// TIA Portal V20 export
DATA_BLOCK "LBP_ParamAlarmMsgs"   // DB5
TITLE = PLC-Error / Messages / Erreur AP / messages
{ S7_Optimized_Access := 'FALSE' }
AUTHOR : SINUMERIK
FAMILY : SINUMERIK_ONE
VERSION : 6.24
// Interface between user program and LBP_GenAlarmMsgs [FC10], contains the parameter assignment of the alarms for the bit arrays in the LBP_AlarmMsgs [DB2] as fault or status message. / Interface entre programme utilisateur et LBP_GenAlarmMsgs [FC10] contient l'affectation de paramètres des alarmes pour les tableaux de bits dans LBP_AlarmMsgs [DB2]  en tant que signalisations de défaut et d'état.
// stored: AutoNumber false
   VAR RETAIN
      Ch1_DB2_310 : Bool := TRUE;   // (Channels 1-10, 18 bits each): DB2.DBB310; error messages / (Canaux 1-10, 18 bits chacun) : DB2.DBB310 ; signalisations de défaut
      Ch1_DB2_311 : Bool := FALSE;   // Channel 1, DB2.DBB311; operating messages / Canal 1, DB2.DBB311 ; signalisations d'état
      Ch1_DB2_312 : Bool := TRUE;   // Channel 1, DB2.DBB312; error messages / Canal 1, DB2.DBB312 ; signalisations de défaut
      Ch1_DB2_313 : Bool := TRUE;   // Error messages / Signalisations de défaut
      Ch1_DB2_314 : Bool := FALSE;   // Operating messages / Signalisations d'état
      Ch1_DB2_315 : Bool := FALSE;   // Operating messages / Signalisations d'état
      Ch1_DB2_316 : Bool := TRUE;   // Error messages / Signalisations de défaut
      Ch1_DB2_317 : Bool := TRUE;   // Error messages / Signalisations de défaut
      Ch1_DB2_318 : Bool := FALSE;   // Operating messages / Signalisations d'état
      Ch1_DB2_319 : Bool := FALSE;   // Operating messages / Signalisations d'état
      Ch1_DB2_320 : Bool := TRUE;   // Error messages / Signalisations de défaut
      Ch1_DB2_321 : Bool := FALSE;   // Operating messages / Signalisations d'état
      Ch1_DB2_322 : Bool := TRUE;   // Error messages / Signalisations de défaut
      Ch1_DB2_323 : Bool := FALSE;   // Operating messages / Signalisations d'état
      Ch1_DB2_324 : Bool := TRUE;   // Error messages / Signalisations de défaut
      Ch1_DB2_325 : Bool := FALSE;   // Operating messages / Signalisations d'état
      Ch1_DB2_326 : Bool := TRUE;   // Error messages / Signalisations de défaut
      Ch1_DB2_327 : Bool := FALSE;   // Operating messages / Signalisations d'état
      Ch2_DB2_328 : Bool := TRUE;   // Channel 2, DB2.DBB328; error messages / Canal 2, DB2.DBB328 ; signalisations de défaut
      Ch2_DB2_329 : Bool := FALSE;   // Channel 2, DB2.DBB329; operating messages / Canal 2, DB2.DBB329 ; signalisations d'état
      Ch2_DB2_330 : Bool := TRUE;   // Error messages / Signalisations de défaut
      Ch2_DB2_331 : Bool := TRUE;   // Error messages / Signalisations de défaut
      Ch2_DB2_332 : Bool := FALSE;   // Operating messages / Signalisations d'état
      Ch2_DB2_333 : Bool := FALSE;   // Operating messages / Signalisations d'état
      Ch2_DB2_334 : Bool := TRUE;   // Error messages / Signalisations de défaut
      Ch2_DB2_335 : Bool := TRUE;   // Error messages / Signalisations de défaut
      Ch2_DB2_336 : Bool := FALSE;   // Operating messages / Signalisations d'état
      Ch2_DB2_337 : Bool := FALSE;   // Operating messages / Signalisations d'état
      Ch2_DB2_338 : Bool := TRUE;   // Error messages / Signalisations de défaut
      Ch2_DB2_339 : Bool := FALSE;   // Operating messages / Signalisations d'état
      Ch2_DB2_340 : Bool := TRUE;   // Error messages / Signalisations de défaut
      Ch2_DB2_341 : Bool := FALSE;   // Operating messages / Signalisations d'état
      Ch2_DB2_342 : Bool := TRUE;   // Error messages / Signalisations de défaut
      Ch2_DB2_343 : Bool := FALSE;   // Operating messages / Signalisations d'état
      Ch2_DB2_344 : Bool := TRUE;   // Error messages / Signalisations de défaut
      Ch2_DB2_345 : Bool := FALSE;   // Operating messages / Signalisations d'état
      Ch3_DB2_346 : Bool := TRUE;   // Channel 3, DB2.DBB346; error messages / Canal 3, DB2.DBB346 ; signalisations de défaut
      Ch3_DB2_347 : Bool := FALSE;   // Channel 3, DB2.DBB347; operating messages / Canal 3, DB2.DBB347 ; signalisations d'état
      Ch3_DB2_348 : Bool := TRUE;   // Error messages / Signalisations de défaut
      Ch3_DB2_349 : Bool := TRUE;   // Error messages / Signalisations de défaut
      Ch3_DB2_350 : Bool := FALSE;   // Operating messages / Signalisations d'état
      Ch3_DB2_351 : Bool := FALSE;   // Operating messages / Signalisations d'état
      Ch3_DB2_352 : Bool := TRUE;   // Error messages / Signalisations de défaut
      Ch3_DB2_353 : Bool := TRUE;   // Error messages / Signalisations de défaut
      Ch3_DB2_354 : Bool := FALSE;   // Operating messages / Signalisations d'état
      Ch3_DB2_355 : Bool := FALSE;   // Operating messages / Signalisations d'état
      Ch3_DB2_356 : Bool := TRUE;   // Error messages / Signalisations de défaut
      Ch3_DB2_357 : Bool := FALSE;   // Operating messages / Signalisations d'état
      Ch3_DB2_358 : Bool := TRUE;   // Error messages / Signalisations de défaut
      Ch3_DB2_359 : Bool := FALSE;   // Operating messages / Signalisations d'état
      Ch3_DB2_360 : Bool := TRUE;   // Error messages / Signalisations de défaut
      Ch3_DB2_361 : Bool := FALSE;   // Operating messages / Signalisations d'état
      Ch3_DB2_362 : Bool := TRUE;   // Error messages / Signalisations de défaut
      Ch3_DB2_363 : Bool := FALSE;   // Operating messages / Signalisations d'état
      Ch4_DB2_364 : Bool := TRUE;   // Channel 4, DB2.DBB364; error messages / Canal 4, DB2.DBB364 ; signalisations de défaut
      Ch4_DB2_365 : Bool := FALSE;   // Channel 4, DB2.DBB365; operating messages / Canal 4, DB2.DBB365 ; signalisations d'état
      Ch4_DB2_366 : Bool := TRUE;   // Error messages / Signalisations de défaut
      Ch4_DB2_367 : Bool := TRUE;   // Error messages / Signalisations de défaut
      Ch4_DB2_368 : Bool := FALSE;   // Operating messages / Signalisations d'état
      Ch4_DB2_369 : Bool := FALSE;   // Operating messages / Signalisations d'état
      Ch4_DB2_370 : Bool := TRUE;   // Error messages / Signalisations de défaut
      Ch4_DB2_371 : Bool := TRUE;   // Error messages / Signalisations de défaut
      Ch4_DB2_372 : Bool := FALSE;   // Operating messages / Signalisations d'état
      Ch4_DB2_373 : Bool := FALSE;   // Operating messages / Signalisations d'état
      Ch4_DB2_374 : Bool := TRUE;   // Error messages / Signalisations de défaut
      Ch4_DB2_375 : Bool := FALSE;   // Operating messages / Signalisations d'état
      Ch4_DB2_376 : Bool := TRUE;   // Error messages / Signalisations de défaut
      Ch4_DB2_377 : Bool := FALSE;   // Operating messages / Signalisations d'état
      Ch4_DB2_378 : Bool := TRUE;   // Error messages / Signalisations de défaut
      Ch4_DB2_379 : Bool := FALSE;   // Operating messages / Signalisations d'état
      Ch4_DB2_380 : Bool := TRUE;   // Error messages / Signalisations de défaut
      Ch4_DB2_381 : Bool := FALSE;   // Operating messages / Signalisations d'état
      Ch5_DB2_382 : Bool := TRUE;   // Channel 5, DB2.DBB382; error messages / Canal 5, DB2.DBB382 ; signalisations de défaut
      Ch5_DB2_383 : Bool := FALSE;   // Channel 5, DB2.DBB383; operating messages / Canal 5, DB2.DBB383 ; signalisations d'état
      Ch5_DB2_384 : Bool := TRUE;   // Error messages / Signalisations de défaut
      Ch5_DB2_385 : Bool := TRUE;   // Error messages / Signalisations de défaut
      Ch5_DB2_386 : Bool := FALSE;   // Operating messages / Signalisations d'état
      Ch5_DB2_387 : Bool := FALSE;   // Operating messages / Signalisations d'état
      Ch5_DB2_388 : Bool := TRUE;   // Error messages / Signalisations de défaut
      Ch5_DB2_389 : Bool := TRUE;   // Error messages / Signalisations de défaut
      Ch5_DB2_390 : Bool := FALSE;   // Operating messages / Signalisations d'état
      Ch5_DB2_391 : Bool := FALSE;   // Operating messages / Signalisations d'état
      Ch5_DB2_392 : Bool := TRUE;   // Error messages / Signalisations de défaut
      Ch5_DB2_393 : Bool := FALSE;   // Operating messages / Signalisations d'état
      Ch5_DB2_394 : Bool := TRUE;   // Error messages / Signalisations de défaut
      Ch5_DB2_395 : Bool := FALSE;   // Operating messages / Signalisations d'état
      Ch5_DB2_396 : Bool := TRUE;   // Error messages / Signalisations de défaut
      Ch5_DB2_397 : Bool := FALSE;   // Operating messages / Signalisations d'état
      Ch5_DB2_398 : Bool := TRUE;   // Error messages / Signalisations de défaut
      Ch5_DB2_399 : Bool := FALSE;   // Operating messages / Signalisations d'état
      Ch6_DB2_400 : Bool := TRUE;   // Channel 6, DB2.DBB400; error messages / Canal 6, DB2.DBB400 ; signalisations de défaut
      Ch6_DB2_401 : Bool := FALSE;   // Channel 6, DB2.DBB401; operating messages / Canal 6, DB2.DBB401 ; signalisations d'état
      Ch6_DB2_402 : Bool := TRUE;   // Error messages / Signalisations de défaut
      Ch6_DB2_403 : Bool := TRUE;   // Error messages / Signalisations de défaut
      Ch6_DB2_404 : Bool := FALSE;   // Operating messages / Signalisations d'état
      Ch6_DB2_405 : Bool := FALSE;   // Operating messages / Signalisations d'état
      Ch6_DB2_406 : Bool := TRUE;   // Error messages / Signalisations de défaut
      Ch6_DB2_407 : Bool := TRUE;   // Error messages / Signalisations de défaut
      Ch6_DB2_408 : Bool := FALSE;   // Operating messages / Signalisations d'état
      Ch6_DB2_409 : Bool := FALSE;   // Operating messages / Signalisations d'état
      Ch6_DB2_410 : Bool := TRUE;   // Error messages / Signalisations de défaut
      Ch6_DB2_411 : Bool := FALSE;   // Operating messages / Signalisations d'état
      Ch6_DB2_412 : Bool := TRUE;   // Error messages / Signalisations de défaut
      Ch6_DB2_413 : Bool := FALSE;   // Operating messages / Signalisations d'état
      Ch6_DB2_414 : Bool := TRUE;   // Error messages / Signalisations de défaut
      Ch6_DB2_415 : Bool := FALSE;   // Operating messages / Signalisations d'état
      Ch6_DB2_416 : Bool := TRUE;   // Error messages / Signalisations de défaut
      Ch6_DB2_417 : Bool := FALSE;   // Operating messages / Signalisations d'état
      Ch7_DB2_418 : Bool := TRUE;   // Channel 7, DB2.DBB418; error messages / Canal 7, DB2.DBB418 ; signalisations de défaut
      Ch7_DB2_419 : Bool := FALSE;   // Channel 7, DB2.DBB419; operating messages / Canal 7, DB2.DBB419 ; signalisations d'état
      Ch7_DB2_420 : Bool := TRUE;   // Error messages / Signalisations de défaut
      Ch7_DB2_421 : Bool := TRUE;   // Error messages / Signalisations de défaut
      Ch7_DB2_422 : Bool := FALSE;   // Operating messages / Signalisations d'état
      Ch7_DB2_423 : Bool := FALSE;   // Operating messages / Signalisations d'état
      Ch7_DB2_424 : Bool := TRUE;   // Error messages / Signalisations de défaut
      Ch7_DB2_425 : Bool := TRUE;   // Error messages / Signalisations de défaut
      Ch7_DB2_426 : Bool := FALSE;   // Operating messages / Signalisations d'état
      Ch7_DB2_427 : Bool := FALSE;   // Operating messages / Signalisations d'état
      Ch7_DB2_428 : Bool := TRUE;   // Error messages / Signalisations de défaut
      Ch7_DB2_429 : Bool := FALSE;   // Operating messages / Signalisations d'état
      Ch7_DB2_430 : Bool := TRUE;   // Error messages / Signalisations de défaut
      Ch7_DB2_431 : Bool := FALSE;   // Operating messages / Signalisations d'état
      Ch7_DB2_432 : Bool := TRUE;   // Error messages / Signalisations de défaut
      Ch7_DB2_433 : Bool := FALSE;   // Operating messages / Signalisations d'état
      Ch7_DB2_434 : Bool := TRUE;   // Error messages / Signalisations de défaut
      Ch7_DB2_435 : Bool := FALSE;   // Operating messages / Signalisations d'état
      Ch8_DB2_436 : Bool := TRUE;   // Channel 8, DB2.DBB436; error messages / Canal 8, DB2.DBB436 ; signalisations de défaut
      Ch8_DB2_437 : Bool := FALSE;   // Channel 8, DB2.DBB437; operating messages / Canal 8, DB2.DBB437 ; signalisations d'état
      Ch8_DB2_438 : Bool := TRUE;   // Error messages / Signalisations de défaut
      Ch8_DB2_439 : Bool := TRUE;   // Error messages / Signalisations de défaut
      Ch8_DB2_440 : Bool := FALSE;   // Operating messages / Signalisations d'état
      Ch8_DB2_441 : Bool := FALSE;   // Operating messages / Signalisations d'état
      Ch8_DB2_442 : Bool := TRUE;   // Error messages / Signalisations de défaut
      Ch8_DB2_443 : Bool := TRUE;   // Error messages / Signalisations de défaut
      Ch8_DB2_444 : Bool := FALSE;   // Operating messages / Signalisations d'état
      Ch8_DB2_445 : Bool := FALSE;   // Operating messages / Signalisations d'état
      Ch8_DB2_446 : Bool := TRUE;   // Error messages / Signalisations de défaut
      Ch8_DB2_447 : Bool := FALSE;   // Operating messages / Signalisations d'état
      Ch8_DB2_448 : Bool := TRUE;   // Error messages / Signalisations de défaut
      Ch8_DB2_449 : Bool := FALSE;   // Operating messages / Signalisations d'état
      Ch8_DB2_450 : Bool := TRUE;   // Error messages / Signalisations de défaut
      Ch8_DB2_451 : Bool := FALSE;   // Operating messages / Signalisations d'état
      Ch8_DB2_452 : Bool := TRUE;   // Error messages / Signalisations de défaut
      Ch8_DB2_453 : Bool := FALSE;   // Operating messages / Signalisations d'état
      Ch9_DB2_454 : Bool := TRUE;   // Channel 9, DB2.DBB454; error messages / Canal 9, DB2.DBB454 ; signalisations de défaut
      Ch9_DB2_455 : Bool := FALSE;   // Channel 9, DB2.DBB455; operating messages / Canal 9, DB2.DBB455 ; signalisations d'état
      Ch9_DB2_456 : Bool := TRUE;   // Error messages / Signalisations de défaut
      Ch9_DB2_457 : Bool := TRUE;   // Error messages / Signalisations de défaut
      Ch9_DB2_458 : Bool := FALSE;   // Operating messages / Signalisations d'état
      Ch9_DB2_459 : Bool := FALSE;   // Operating messages / Signalisations d'état
      Ch9_DB2_460 : Bool := TRUE;   // Error messages / Signalisations de défaut
      Ch9_DB2_461 : Bool := TRUE;   // Error messages / Signalisations de défaut
      Ch9_DB2_462 : Bool := FALSE;   // Operating messages / Signalisations d'état
      Ch9_DB2_463 : Bool := FALSE;   // Operating messages / Signalisations d'état
      Ch9_DB2_464 : Bool := TRUE;   // Error messages / Signalisations de défaut
      Ch9_DB2_465 : Bool := FALSE;   // Operating messages / Signalisations d'état
      Ch9_DB2_466 : Bool := TRUE;   // Error messages / Signalisations de défaut
      Ch9_DB2_467 : Bool := FALSE;   // Operating messages / Signalisations d'état
      Ch9_DB2_468 : Bool := TRUE;   // Error messages / Signalisations de défaut
      Ch9_DB2_469 : Bool := FALSE;   // Operating messages / Signalisations d'état
      Ch9_DB2_470 : Bool := TRUE;   // Error messages / Signalisations de défaut
      Ch9_DB2_471 : Bool := FALSE;   // Operating messages / Signalisations d'état
      Ch10_DB2_472 : Bool := TRUE;   // Channel 10, DB2.DBB472; error messages / Canal 10, DB2.DBB472 ; signalisations de défaut
      Ch10_DB2_473 : Bool := FALSE;   // Channel 10, DB2.DBB473; operating messages / Canal 10, DB2.DBB473 ; signalisations d'état
      Ch10_DB2_474 : Bool := TRUE;   // Error messages / Signalisations de défaut
      Ch10_DB2_475 : Bool := TRUE;   // Error messages / Signalisations de défaut
      Ch10_DB2_476 : Bool := FALSE;   // Operating messages / Signalisations d'état
      Ch10_DB2_477 : Bool := FALSE;   // Operating messages / Signalisations d'état
      Ch10_DB2_478 : Bool := TRUE;   // Error messages / Signalisations de défaut
      Ch10_DB2_479 : Bool := TRUE;   // Error messages / Signalisations de défaut
      Ch10_DB2_480 : Bool := FALSE;   // Operating messages / Signalisations d'état
      Ch10_DB2_481 : Bool := FALSE;   // Operating messages / Signalisations d'état
      Ch10_DB2_482 : Bool := TRUE;   // Error messages / Signalisations de défaut
      Ch10_DB2_483 : Bool := FALSE;   // Operating messages / Signalisations d'état
      Ch10_DB2_484 : Bool := TRUE;   // Error messages / Signalisations de défaut
      Ch10_DB2_485 : Bool := FALSE;   // Operating messages / Signalisations d'état
      Ch10_DB2_486 : Bool := TRUE;   // Error messages / Signalisations de défaut
      Ch10_DB2_487 : Bool := FALSE;   // Operating messages / Signalisations d'état
      Ch10_DB2_488 : Bool := TRUE;   // Error messages / Signalisations de défaut
      Ch10_DB2_489 : Bool := FALSE;   // Operating messages / Signalisations d'état
      Ax1_DB2_490 : Bool := TRUE;   // (Axes/Spindles 1-31, 2 bits each): DB2.DBB490; error messages / (Axes/broches 1-31, 2 bits chacun) : DB2.DBB490 ; signalisations de défaut
      Ax1_DB2_491 : Bool := FALSE;   // Axis/Spindle 1, DB2.DBB491; operating messages / Axe/broche 1, DB2.DBB491 ; signalisations d'état
      Ax2_DB2_492 : Bool := TRUE;   // Axis/Spindle 2, DB2.DBB492; error messages / Axe/broche 2, DB2.DBB492 ; signalisations de défaut
      Ax2_DB2_493 : Bool := FALSE;   // Axis/Spindle 2, DB2.DBB493; operating messages / Axe/broche 2, DB2.DBB493 ; signalisations d'état
      Ax3_DB2_494 : Bool := TRUE;   // Error messages / Signalisations de défaut
      Ax3_DB2_495 : Bool := FALSE;   // Operating messages / Signalisations d'état
      Ax4_DB2_496 : Bool := TRUE;   // Error messages / Signalisations de défaut
      Ax4_DB2_497 : Bool := FALSE;   // Operating messages / Signalisations d'état
      Ax5_DB2_498 : Bool := TRUE;   // Error messages / Signalisations de défaut
      Ax5_DB2_499 : Bool := FALSE;   // Operating messages / Signalisations d'état
      Ax6_DB2_500 : Bool := TRUE;   // Error messages / Signalisations de défaut
      Ax6_DB2_501 : Bool := FALSE;   // Operating messages / Signalisations d'état
      Ax7_DB2_502 : Bool := TRUE;   // Error messages / Signalisations de défaut
      Ax7_DB2_503 : Bool := FALSE;   // Operating messages / Signalisations d'état
      Ax8_DB2_504 : Bool := TRUE;   // Error messages / Signalisations de défaut
      Ax8_DB2_505 : Bool := FALSE;   // Operating messages / Signalisations d'état
      Ax9_DB2_506 : Bool := TRUE;   // Error messages / Signalisations de défaut
      Ax9_DB2_507 : Bool := FALSE;   // Operating messages / Signalisations d'état
      Ax10_DB2_508 : Bool := TRUE;   // Error messages / Signalisations de défaut
      Ax10_DB2_509 : Bool := FALSE;   // Operating messages / Signalisations d'état
      Ax11_DB2_510 : Bool := TRUE;   // Error messages / Signalisations de défaut
      Ax11_DB2_511 : Bool := FALSE;   // Operating messages / Signalisations d'état
      Ax12_DB2_512 : Bool := TRUE;   // Error messages / Signalisations de défaut
      Ax12_DB2_513 : Bool := FALSE;   // Operating messages / Signalisations d'état
      Ax13_DB2_514 : Bool := TRUE;   // Error messages / Signalisations de défaut
      Ax13_DB2_515 : Bool := FALSE;   // Operating messages / Signalisations d'état
      Ax14_DB2_516 : Bool := TRUE;   // Error messages / Signalisations de défaut
      Ax14_DB2_517 : Bool := FALSE;   // Operating messages / Signalisations d'état
      Ax15_DB2_518 : Bool := TRUE;   // Error messages / Signalisations de défaut
      Ax15_DB2_519 : Bool := FALSE;   // Operating messages / Signalisations d'état
      Ax16_DB2_520 : Bool := TRUE;   // Error messages / Signalisations de défaut
      Ax16_DB2_521 : Bool := FALSE;   // Operating messages / Signalisations d'état
      Ax17_DB2_522 : Bool := TRUE;   // Error messages / Signalisations de défaut
      Ax17_DB2_523 : Bool := FALSE;   // Operating messages / Signalisations d'état
      Ax18_DB2_524 : Bool := TRUE;   // Error messages / Signalisations de défaut
      Ax18_DB2_525 : Bool := FALSE;   // Operating messages / Signalisations d'état
      Ax19_DB2_526 : Bool := TRUE;   // Error messages / Signalisations de défaut
      Ax19_DB2_527 : Bool := FALSE;   // Operating messages / Signalisations d'état
      Ax20_DB2_528 : Bool := TRUE;   // Error messages / Signalisations de défaut
      Ax20_DB2_529 : Bool := FALSE;   // Operating messages / Signalisations d'état
      Ax21_DB2_530 : Bool := TRUE;   // Error messages / Signalisations de défaut
      Ax21_DB2_531 : Bool := FALSE;   // Operating messages / Signalisations d'état
      Ax22_DB2_532 : Bool := TRUE;   // Error messages / Signalisations de défaut
      Ax22_DB2_533 : Bool := FALSE;   // Operating messages / Signalisations d'état
      Ax23_DB2_534 : Bool := TRUE;   // Error messages / Signalisations de défaut
      Ax23_DB2_535 : Bool := FALSE;   // Operating messages / Signalisations d'état
      Ax24_DB2_536 : Bool := TRUE;   // Error messages / Signalisations de défaut
      Ax24_DB2_537 : Bool := FALSE;   // Operating messages / Signalisations d'état
      Ax25_DB2_538 : Bool := TRUE;   // Error messages / Signalisations de défaut
      Ax25_DB2_539 : Bool := FALSE;   // Operating messages / Signalisations d'état
      Ax26_DB2_540 : Bool := TRUE;   // Error messages / Signalisations de défaut
      Ax26_DB2_541 : Bool := FALSE;   // Operating messages / Signalisations d'état
      Ax27_DB2_542 : Bool := TRUE;   // Error messages / Signalisations de défaut
      Ax27_DB2_543 : Bool := FALSE;   // Operating messages / Signalisations d'état
      Ax28_DB2_544 : Bool := TRUE;   // Error messages / Signalisations de défaut
      Ax28_DB2_545 : Bool := FALSE;   // Operating messages / Signalisations d'état
      Ax29_DB2_546 : Bool := TRUE;   // Error messages / Signalisations de défaut
      Ax29_DB2_547 : Bool := FALSE;   // Operating messages / Signalisations d'état
      Ax30_DB2_548 : Bool := TRUE;   // Error messages / Signalisations de défaut
      Ax30_DB2_549 : Bool := FALSE;   // Operating messages / Signalisations d'état
      Ax31_DB2_550 : Bool := TRUE;   // Error messages / Signalisations de défaut
      Ax31_DB2_551 : Bool := FALSE;   // Operating messages / Signalisations d'état
      Bit30_2 : Bool := FALSE;   // Reserved / Réservé
      Bit30_3 : Bool := FALSE;   // Reserved / Réservé
      User0_DB2_554 : Bool := TRUE;   // (User data areas 0-31, 8 bits each): DB2.DBB554; error messages / (Zones de donnés utilisateur 0-31, 8 bits chacune) : DB2.DBB554 ; signalisations de défaut
      User0_DB2_555 : Bool := TRUE;   // UserDataArea 0, DB2.DBB555; error messages / UserDataArea 0, DB2.DBB555 ; signalisations de défaut
      User0_DB2_556 : Bool := TRUE;   // Error messages / Signalisations de défaut
      User0_DB2_557 : Bool := TRUE;   // Error messages / Signalisations de défaut
      User0_DB2_558 : Bool := FALSE;   // Operating messages / Signalisations d'état
      User0_DB2_559 : Bool := FALSE;   // Operating messages / Signalisations d'état
      User0_DB2_560 : Bool := FALSE;   // Operating messages / Signalisations d'état
      User0_DB2_561 : Bool := FALSE;   // Operating messages / Signalisations d'état
      User1_DB2_562 : Bool := TRUE;   // UserDataArea 1, DB2.DBB562; error messages / UserDataArea 1, DB2.DBB562 ; signalisations de défaut
      User1_DB2_563 : Bool := TRUE;   // Error messages / Signalisations de défaut
      User1_DB2_564 : Bool := TRUE;   // Error messages / Signalisations de défaut
      User1_DB2_565 : Bool := TRUE;   // Error messages / Signalisations de défaut
      User1_DB2_566 : Bool := FALSE;   // Operating messages / Signalisations d'état
      User1_DB2_567 : Bool := FALSE;   // Operating messages / Signalisations d'état
      User1_DB2_568 : Bool := FALSE;   // Operating messages / Signalisations d'état
      User1_DB2_569 : Bool := FALSE;   // Operating messages / Signalisations d'état
      User2_DB2_570 : Bool := TRUE;   // UserDataArea 2, DB2.DBB570; error messages / UserDataArea 2, DB2.DBB570 ; signalisations de défaut
      User2_DB2_571 : Bool := TRUE;   // Error messages / Signalisations de défaut
      User2_DB2_572 : Bool := TRUE;   // Error messages / Signalisations de défaut
      User2_DB2_573 : Bool := TRUE;   // Error messages / Signalisations de défaut
      User2_DB2_574 : Bool := FALSE;   // Operating messages / Signalisations d'état
      User2_DB2_575 : Bool := FALSE;   // Operating messages / Signalisations d'état
      User2_DB2_576 : Bool := FALSE;   // Operating messages / Signalisations d'état
      User2_DB2_577 : Bool := FALSE;   // Operating messages / Signalisations d'état
      User3_DB2_578 : Bool := TRUE;   // UserDataArea 3, DB2.DBB578; error messages / UserDataArea 3, DB2.DBB578 ; signalisations de défaut
      User3_DB2_579 : Bool := TRUE;   // Error messages / Signalisations de défaut
      User3_DB2_580 : Bool := TRUE;   // Error messages / Signalisations de défaut
      User3_DB2_581 : Bool := TRUE;   // Error messages / Signalisations de défaut
      User3_DB2_582 : Bool := FALSE;   // Operating messages / Signalisations d'état
      User3_DB2_583 : Bool := FALSE;   // Operating messages / Signalisations d'état
      User3_DB2_584 : Bool := FALSE;   // Operating messages / Signalisations d'état
      User3_DB2_585 : Bool := FALSE;   // Operating messages / Signalisations d'état
      User4_DB2_586 : Bool := TRUE;   // UserDataArea 4, DB2.DBB586; error messages / UserDataArea 4, DB2.DBB586 ; signalisations de défaut
      User4_DB2_587 : Bool := TRUE;   // Error messages / Signalisations de défaut
      User4_DB2_588 : Bool := TRUE;   // Error messages / Signalisations de défaut
      User4_DB2_589 : Bool := TRUE;   // Error messages / Signalisations de défaut
      User4_DB2_590 : Bool := FALSE;   // Operating messages / Signalisations d'état
      User4_DB2_591 : Bool := FALSE;   // Operating messages / Signalisations d'état
      User4_DB2_592 : Bool := FALSE;   // Operating messages / Signalisations d'état
      User4_DB2_593 : Bool := FALSE;   // Operating messages / Signalisations d'état
      User5_DB2_594 : Bool := TRUE;   // UserDataArea 5, DB2.DBB594; error messages / UserDataArea 5, DB2.DBB594 ; signalisations de défaut
      User5_DB2_595 : Bool := TRUE;   // Error messages / Signalisations de défaut
      User5_DB2_596 : Bool := TRUE;   // Error messages / Signalisations de défaut
      User5_DB2_597 : Bool := TRUE;   // Error messages / Signalisations de défaut
      User5_DB2_598 : Bool := FALSE;   // Operating messages / Signalisations d'état
      User5_DB2_599 : Bool := FALSE;   // Operating messages / Signalisations d'état
      User5_DB2_600 : Bool := FALSE;   // Operating messages / Signalisations d'état
      User5_DB2_601 : Bool := FALSE;   // Operating messages / Signalisations d'état
      User6_DB2_602 : Bool := TRUE;   // UserDataArea 6, DB2.DBB602; error messages / UserDataArea 6, DB2.DBB602 ; signalisations de défaut
      User6_DB2_603 : Bool := TRUE;   // Error messages / Signalisations de défaut
      User6_DB2_604 : Bool := TRUE;   // Error messages / Signalisations de défaut
      User6_DB2_605 : Bool := TRUE;   // Error messages / Signalisations de défaut
      User6_DB2_606 : Bool := FALSE;   // Operating messages / Signalisations d'état
      User6_DB2_607 : Bool := TRUE;   // Operating messages / Signalisations d'état
      User6_DB2_608 : Bool := TRUE;   // Operating messages / Signalisations d'état
      User6_DB2_609 : Bool := TRUE;   // Operating messages / Signalisations d'état
      User7_DB2_610 : Bool := FALSE;   // UserDataArea 7, DB2.DBB610; error messages / UserDataArea 7, DB2.DBB610 ; signalisations de défaut
      User7_DB2_611 : Bool := FALSE;   // Error messages / Signalisations de défaut
      User7_DB2_612 : Bool := FALSE;   // Error messages / Signalisations de défaut
      User7_DB2_613 : Bool := FALSE;   // Error messages / Signalisations de défaut
      User7_DB2_614 : Bool := FALSE;   // Operating messages / Signalisations d'état
      User7_DB2_615 : Bool := FALSE;   // Operating messages / Signalisations d'état
      User7_DB2_616 : Bool := FALSE;   // Operating messages / Signalisations d'état
      User7_DB2_617 : Bool := FALSE;   // Operating messages / Signalisations d'état
      User8_DB2_618 : Bool := TRUE;   // UserDataArea 8, DB2.DBB618; error messages / UserDataArea 8, DB2.DBB618 ; signalisations de défaut
      User8_DB2_619 : Bool := TRUE;   // Error messages / Signalisations de défaut
      User8_DB2_620 : Bool := TRUE;   // Error messages / Signalisations de défaut
      User8_DB2_621 : Bool := TRUE;   // Error messages / Signalisations de défaut
      User8_DB2_622 : Bool := FALSE;   // Operating messages / Signalisations d'état
      User8_DB2_623 : Bool := FALSE;   // Operating messages / Signalisations d'état
      User8_DB2_624 : Bool := FALSE;   // Operating messages / Signalisations d'état
      User8_DB2_625 : Bool := FALSE;   // Operating messages / Signalisations d'état
      User9_DB2_626 : Bool := TRUE;   // UserDataArea 9, DB2.DBB626; error messages / UserDataArea 9, DB2.DBB626 ; signalisations de défaut
      User9_DB2_627 : Bool := TRUE;   // Error messages / Signalisations de défaut
      User9_DB2_628 : Bool := TRUE;   // Error messages / Signalisations de défaut
      User9_DB2_629 : Bool := TRUE;   // Error messages / Signalisations de défaut
      User9_DB2_630 : Bool := FALSE;   // Operating messages / Signalisations d'état
      User9_DB2_631 : Bool := FALSE;   // Operating messages / Signalisations d'état
      User9_DB2_632 : Bool := FALSE;   // Operating messages / Signalisations d'état
      User9_DB2_633 : Bool := FALSE;   // Operating messages / Signalisations d'état
      User10_DB2_634 : Bool := TRUE;   // UserDataArea 10, DB2.DBB634; error messages / UserDataArea 10, DB2.DBB634 ; signalisations de défaut
      User10_DB2_635 : Bool := TRUE;   // Error messages / Signalisations de défaut
      User10_DB2_636 : Bool := TRUE;   // Error messages / Signalisations de défaut
      User10_DB2_637 : Bool := TRUE;   // Error messages / Signalisations de défaut
      User10_DB2_638 : Bool := FALSE;   // Operating messages / Signalisations d'état
      User10_DB2_639 : Bool := FALSE;   // Operating messages / Signalisations d'état
      User10_DB2_640 : Bool := FALSE;   // Operating messages / Signalisations d'état
      User10_DB2_641 : Bool := FALSE;   // Operating messages / Signalisations d'état
      User11_DB2_642 : Bool := TRUE;   // UserDataArea 11, DB2.DBB642; error messages / UserDataArea 11, DB2.DBB642 ; signalisations de défaut
      User11_DB2_643 : Bool := TRUE;   // Error messages / Signalisations de défaut
      User11_DB2_644 : Bool := TRUE;   // Error messages / Signalisations de défaut
      User11_DB2_645 : Bool := TRUE;   // Error messages / Signalisations de défaut
      User11_DB2_646 : Bool := FALSE;   // Operating messages / Signalisations d'état
      User11_DB2_647 : Bool := FALSE;   // Operating messages / Signalisations d'état
      User11_DB2_648 : Bool := FALSE;   // Operating messages / Signalisations d'état
      User11_DB2_649 : Bool := FALSE;   // Operating messages / Signalisations d'état
      User12_DB2_650 : Bool := TRUE;   // UserDataArea 12, DB2.DBB650; error messages / UserDataArea 12, DB2.DBB650 ; signalisations de défaut
      User12_DB2_651 : Bool := TRUE;   // Error messages / Signalisations de défaut
      User12_DB2_652 : Bool := TRUE;   // Error messages / Signalisations de défaut
      User12_DB2_653 : Bool := TRUE;   // Error messages / Signalisations de défaut
      User12_DB2_654 : Bool := FALSE;   // Operating messages / Signalisations d'état
      User12_DB2_655 : Bool := FALSE;   // Operating messages / Signalisations d'état
      User12_DB2_656 : Bool := FALSE;   // Operating messages / Signalisations d'état
      User12_DB2_657 : Bool := FALSE;   // Operating messages / Signalisations d'état
      User13_DB2_658 : Bool := TRUE;   // UserDataArea 13, DB2.DBB658; error messages / UserDataArea 13, DB2.DBB658 ; signalisations de défaut
      User13_DB2_659 : Bool := TRUE;   // Error messages / Signalisations de défaut
      User13_DB2_660 : Bool := TRUE;   // Error messages / Signalisations de défaut
      User13_DB2_661 : Bool := TRUE;   // Error messages / Signalisations de défaut
      User13_DB2_662 : Bool := FALSE;   // Operating messages / Signalisations d'état
      User13_DB2_663 : Bool := FALSE;   // Operating messages / Signalisations d'état
      User13_DB2_664 : Bool := FALSE;   // Operating messages / Signalisations d'état
      User13_DB2_665 : Bool := FALSE;   // Operating messages / Signalisations d'état
      User14_DB2_666 : Bool := TRUE;   // UserDataArea 14, DB2.DBB666; error messages / UserDataArea 14, DB2.DBB666 ; signalisations de défaut
      User14_DB2_667 : Bool := TRUE;   // Error messages / Signalisations de défaut
      User14_DB2_668 : Bool := TRUE;   // Error messages / Signalisations de défaut
      User14_DB2_669 : Bool := TRUE;   // Error messages / Signalisations de défaut
      User14_DB2_670 : Bool := FALSE;   // Operating messages / Signalisations d'état
      User14_DB2_671 : Bool := FALSE;   // Operating messages / Signalisations d'état
      User14_DB2_672 : Bool := FALSE;   // Operating messages / Signalisations d'état
      User14_DB2_673 : Bool := FALSE;   // Operating messages / Signalisations d'état
      User15_DB2_674 : Bool := TRUE;   // UserDataArea 15, DB2.DBB674; error messages / UserDataArea 15, DB2.DBB674 ; signalisations de défaut
      User15_DB2_675 : Bool := TRUE;   // Error messages / Signalisations de défaut
      User15_DB2_676 : Bool := TRUE;   // Error messages / Signalisations de défaut
      User15_DB2_677 : Bool := TRUE;   // Error messages / Signalisations de défaut
      User15_DB2_678 : Bool := FALSE;   // Operating messages / Signalisations d'état
      User15_DB2_679 : Bool := FALSE;   // Operating messages / Signalisations d'état
      User15_DB2_680 : Bool := FALSE;   // Operating messages / Signalisations d'état
      User15_DB2_681 : Bool := FALSE;   // Operating messages / Signalisations d'état
      User16_DB2_682 : Bool := TRUE;   // UserDataArea 16, DB2.DBB682; error messages / UserDataArea 16, DB2.DBB682 ; signalisations de défaut
      User16_DB2_683 : Bool := TRUE;   // Error messages / Signalisations de défaut
      User16_DB2_684 : Bool := TRUE;   // Error messages / Signalisations de défaut
      User16_DB2_685 : Bool := TRUE;   // Error messages / Signalisations de défaut
      User16_DB2_686 : Bool := FALSE;   // Operating messages / Signalisations d'état
      User16_DB2_687 : Bool := FALSE;   // Operating messages / Signalisations d'état
      User16_DB2_688 : Bool := FALSE;   // Operating messages / Signalisations d'état
      User16_DB2_689 : Bool := FALSE;   // Operating messages / Signalisations d'état
      User17_DB2_690 : Bool := TRUE;   // UserDataArea 17, DB2.DBB690; error messages / UserDataArea 17, DB2.DBB690 ; signalisations de défaut
      User17_DB2_691 : Bool := TRUE;   // Error messages / Signalisations de défaut
      User17_DB2_692 : Bool := TRUE;   // Error messages / Signalisations de défaut
      User17_DB2_693 : Bool := TRUE;   // Error messages / Signalisations de défaut
      User17_DB2_694 : Bool := FALSE;   // Operating messages / Signalisations d'état
      User17_DB2_695 : Bool := FALSE;   // Operating messages / Signalisations d'état
      User17_DB2_696 : Bool := FALSE;   // Operating messages / Signalisations d'état
      User17_DB2_697 : Bool := FALSE;   // Operating messages / Signalisations d'état
      User18_DB2_698 : Bool := TRUE;   // UserDataArea 18, DB2.DBB698; error messages / UserDataArea 18, DB2.DBB698 ; signalisations de défaut
      User18_DB2_699 : Bool := TRUE;   // Error messages / Signalisations de défaut
      User18_DB2_700 : Bool := TRUE;   // Error messages / Signalisations de défaut
      User18_DB2_701 : Bool := TRUE;   // Error messages / Signalisations de défaut
      User18_DB2_702 : Bool := FALSE;   // Operating messages / Signalisations d'état
      User18_DB2_703 : Bool := FALSE;   // Operating messages / Signalisations d'état
      User18_DB2_704 : Bool := FALSE;   // Operating messages / Signalisations d'état
      User18_DB2_705 : Bool := FALSE;   // Operating messages / Signalisations d'état
      User19_DB2_706 : Bool := TRUE;   // UserDataArea 19, DB2.DBB706; error messages / UserDataArea 19, DB2.DBB706 ; signalisations de défaut
      User19_DB2_707 : Bool := TRUE;   // Error messages / Signalisations de défaut
      User19_DB2_708 : Bool := TRUE;   // Error messages / Signalisations de défaut
      User19_DB2_709 : Bool := TRUE;   // Error messages / Signalisations de défaut
      User19_DB2_710 : Bool := FALSE;   // Operating messages / Signalisations d'état
      User19_DB2_711 : Bool := FALSE;   // Operating messages / Signalisations d'état
      User19_DB2_712 : Bool := FALSE;   // Operating messages / Signalisations d'état
      User19_DB2_713 : Bool := FALSE;   // Operating messages / Signalisations d'état
      User20_DB2_714 : Bool := TRUE;   // UserDataArea 20, DB2.DBB714; error messages / UserDataArea 20, DB2.DBB714 ; signalisations de défaut
      User20_DB2_715 : Bool := TRUE;   // Error messages / Signalisations de défaut
      User20_DB2_716 : Bool := TRUE;   // Error messages / Signalisations de défaut
      User20_DB2_717 : Bool := TRUE;   // Error messages / Signalisations de défaut
      User20_DB2_718 : Bool := FALSE;   // Operating messages / Signalisations d'état
      User20_DB2_719 : Bool := FALSE;   // Operating messages / Signalisations d'état
      User20_DB2_720 : Bool := FALSE;   // Operating messages / Signalisations d'état
      User20_DB2_721 : Bool := FALSE;   // Operating messages / Signalisations d'état
      User21_DB2_722 : Bool := TRUE;   // UserDataArea 21, DB2.DBB722; error messages / UserDataArea 21, DB2.DBB722 ; signalisations de défaut
      User21_DB2_723 : Bool := TRUE;   // Error messages / Signalisations de défaut
      User21_DB2_724 : Bool := TRUE;   // Error messages / Signalisations de défaut
      User21_DB2_725 : Bool := TRUE;   // Error messages / Signalisations de défaut
      User21_DB2_726 : Bool := FALSE;   // Operating messages / Signalisations d'état
      User21_DB2_727 : Bool := FALSE;   // Operating messages / Signalisations d'état
      User21_DB2_728 : Bool := FALSE;   // Operating messages / Signalisations d'état
      User21_DB2_729 : Bool := FALSE;   // Operating messages / Signalisations d'état
      User22_DB2_730 : Bool := TRUE;   // UserDataArea 22, DB2.DBB730; error messages / UserDataArea 22, DB2.DBB730 ; signalisations de défaut
      User22_DB2_731 : Bool := TRUE;   // Error messages / Signalisations de défaut
      User22_DB2_732 : Bool := TRUE;   // Error messages / Signalisations de défaut
      User22_DB2_733 : Bool := TRUE;   // Error messages / Signalisations de défaut
      User22_DB2_734 : Bool := FALSE;   // Operating messages / Signalisations d'état
      User22_DB2_735 : Bool := FALSE;   // Operating messages / Signalisations d'état
      User22_DB2_736 : Bool := FALSE;   // Operating messages / Signalisations d'état
      User22_DB2_737 : Bool := FALSE;   // Operating messages / Signalisations d'état
      User23_DB2_738 : Bool := TRUE;   // UserDataArea 23, DB2.DBB738; error messages / UserDataArea 23, DB2.DBB738 ; signalisations de défaut
      User23_DB2_739 : Bool := TRUE;   // Error messages / Signalisations de défaut
      User23_DB2_740 : Bool := TRUE;   // Error messages / Signalisations de défaut
      User23_DB2_741 : Bool := TRUE;   // Error messages / Signalisations de défaut
      User23_DB2_742 : Bool := FALSE;   // Operating messages / Signalisations d'état
      User23_DB2_743 : Bool := FALSE;   // Operating messages / Signalisations d'état
      User23_DB2_744 : Bool := FALSE;   // Operating messages / Signalisations d'état
      User23_DB2_745 : Bool := FALSE;   // Operating messages / Signalisations d'état
      User24_DB2_746 : Bool := TRUE;   // UserDataArea 24, DB2.DBB746; error messages / UserDataArea 24, DB2.DBB746 ; signalisations de défaut
      User24_DB2_747 : Bool := TRUE;   // Error messages / Signalisations de défaut
      User24_DB2_748 : Bool := TRUE;   // Error messages / Signalisations de défaut
      User24_DB2_749 : Bool := TRUE;   // Error messages / Signalisations de défaut
      User24_DB2_750 : Bool := FALSE;   // Operating messages / Signalisations d'état
      User24_DB2_751 : Bool := FALSE;   // Operating messages / Signalisations d'état
      User24_DB2_752 : Bool := FALSE;   // Operating messages / Signalisations d'état
      User24_DB2_753 : Bool := FALSE;   // Operating messages / Signalisations d'état
      User25_DB2_754 : Bool := TRUE;   // UserDataArea 25, DB2.DBB754; error messages / UserDataArea 25, DB2.DBB754 ; signalisations de défaut
      User25_DB2_755 : Bool := TRUE;   // Error messages / Signalisations de défaut
      User25_DB2_756 : Bool := TRUE;   // Error messages / Signalisations de défaut
      User25_DB2_757 : Bool := TRUE;   // Error messages / Signalisations de défaut
      User25_DB2_758 : Bool := FALSE;   // Operating messages / Signalisations d'état
      User25_DB2_759 : Bool := FALSE;   // Operating messages / Signalisations d'état
      User25_DB2_760 : Bool := FALSE;   // Operating messages / Signalisations d'état
      User25_DB2_761 : Bool := FALSE;   // Operating messages / Signalisations d'état
      User26_DB2_762 : Bool := TRUE;   // UserDataArea 26, DB2.DBB762; error messages / UserDataArea 26, DB2.DBB762 ; signalisations de défaut
      User26_DB2_763 : Bool := TRUE;   // Error messages / Signalisations de défaut
      User26_DB2_764 : Bool := TRUE;   // Error messages / Signalisations de défaut
      User26_DB2_765 : Bool := TRUE;   // Error messages / Signalisations de défaut
      User26_DB2_766 : Bool := FALSE;   // Operating messages / Signalisations d'état
      User26_DB2_767 : Bool := FALSE;   // Operating messages / Signalisations d'état
      User26_DB2_768 : Bool := FALSE;   // Operating messages / Signalisations d'état
      User26_DB2_769 : Bool := FALSE;   // Operating messages / Signalisations d'état
      User27_DB2_770 : Bool := TRUE;   // UserDataArea 27, DB2.DBB770; error messages / UserDataArea 27, DB2.DBB770 ; signalisations de défaut
      User27_DB2_771 : Bool := TRUE;   // Error messages / Signalisations de défaut
      User27_DB2_772 : Bool := TRUE;   // Error messages / Signalisations de défaut
      User27_DB2_773 : Bool := TRUE;   // Error messages / Signalisations de défaut
      User27_DB2_774 : Bool := FALSE;   // Operating messages / Signalisations d'état
      User27_DB2_775 : Bool := FALSE;   // Operating messages / Signalisations d'état
      User27_DB2_776 : Bool := FALSE;   // Operating messages / Signalisations d'état
      User27_DB2_777 : Bool := FALSE;   // Operating messages / Signalisations d'état
      User28_DB2_778 : Bool := TRUE;   // UserDataArea 28, DB2.DBB778; error messages / UserDataArea 28, DB2.DBB778 ; signalisations de défaut
      User28_DB2_779 : Bool := TRUE;   // Error messages / Signalisations de défaut
      User28_DB2_780 : Bool := TRUE;   // Error messages / Signalisations de défaut
      User28_DB2_781 : Bool := TRUE;   // Error messages / Signalisations de défaut
      User28_DB2_782 : Bool := FALSE;   // Operating messages / Signalisations d'état
      User28_DB2_783 : Bool := FALSE;   // Operating messages / Signalisations d'état
      User28_DB2_784 : Bool := FALSE;   // Operating messages / Signalisations d'état
      User28_DB2_785 : Bool := FALSE;   // Operating messages / Signalisations d'état
      User29_DB2_786 : Bool := TRUE;   // UserDataArea 29, DB2.DBB786; error messages / UserDataArea 29, DB2.DBB786 ; signalisations de défaut
      User29_DB2_787 : Bool := TRUE;   // Error messages / Signalisations de défaut
      User29_DB2_788 : Bool := TRUE;   // Error messages / Signalisations de défaut
      User29_DB2_789 : Bool := TRUE;   // Error messages / Signalisations de défaut
      User29_DB2_790 : Bool := FALSE;   // Operating messages / Signalisations d'état
      User29_DB2_791 : Bool := FALSE;   // Operating messages / Signalisations d'état
      User29_DB2_792 : Bool := FALSE;   // Operating messages / Signalisations d'état
      User29_DB2_793 : Bool := FALSE;   // Operating messages / Signalisations d'état
      User30_DB2_794 : Bool := TRUE;   // UserDataArea 30, DB2.DBB794; error messages / UserDataArea 30, DB2.DBB794 ; signalisations de défaut
      User30_DB2_795 : Bool := TRUE;   // Error messages / Signalisations de défaut
      User30_DB2_796 : Bool := TRUE;   // Error messages / Signalisations de défaut
      User30_DB2_797 : Bool := TRUE;   // Error messages / Signalisations de défaut
      User30_DB2_798 : Bool := FALSE;   // Operating messages / Signalisations d'état
      User30_DB2_799 : Bool := FALSE;   // Operating messages / Signalisations d'état
      User30_DB2_800 : Bool := FALSE;   // Operating messages / Signalisations d'état
      User30_DB2_801 : Bool := FALSE;   // Operating messages / Signalisations d'état
      User31_DB2_802 : Bool := TRUE;   // UserDataArea 31, DB2.DBB802; error messages / UserDataArea 31, DB2.DBB802 ; signalisations de défaut
      User31_DB2_803 : Bool := TRUE;   // Error messages / Signalisations de défaut
      User31_DB2_804 : Bool := TRUE;   // Error messages / Signalisations de défaut
      User31_DB2_805 : Bool := TRUE;   // Error messages / Signalisations de défaut
      User31_DB2_806 : Bool := FALSE;   // Operating messages / Signalisations d'état
      User31_DB2_807 : Bool := FALSE;   // Operating messages / Signalisations d'état
      User31_DB2_808 : Bool := FALSE;   // Operating messages / Signalisations d'état
      User31_DB2_809 : Bool := FALSE;   // Operating messages / Signalisations d'état
      Bit62_4 : Bool;   // Reserved / Réservé
      Bit62_5 : Bool;   // Reserved / Réservé
      Bit62_6 : Bool;   // Reserved / Réservé
      Bit62_7 : Bool;   // Reserved / Réservé
      Byte63 : Byte;   // Reserved / Réservé
      Word64 : Word;   // Reserved / Réservé
      Word66 : Word;   // Reserved / Réservé
      Word68 : Word;   // Reserved / Réservé
      Word70 : Word;   // Reserved / Réservé
      ByteArray72 : Array[0..63] of Byte;   // Reserved / Réservé
      User32_DB2_810 : Bool := TRUE;   // (User data areas 32-63, 8 bits each): DB2.DBB810; error messages / (Zones de donnés utilisateur 32-63, 8 bits chacune): DB2.DBB810 ; signalisations de défaut
      User32_DB2_811 : Bool := TRUE;   // Error messages / Signalisations de défaut
      User32_DB2_812 : Bool := TRUE;   // Error messages / Signalisations de défaut
      User32_DB2_813 : Bool := TRUE;   // Error messages / Signalisations de défaut
      User32_DB2_814 : Bool := FALSE;   // Operating messages / Signalisations d'état
      User32_DB2_815 : Bool := FALSE;   // Operating messages / Signalisations d'état
      User32_DB2_816 : Bool := FALSE;   // Operating messages / Signalisations d'état
      User32_DB2_817 : Bool := FALSE;   // Operating messages / Signalisations d'état
      User33_DB2_818 : Bool := TRUE;   // UserDataArea 33, DB2.DBB818; error messages / UserDataArea 33, DB2.DBB818 ; signalisations de défaut
      User33_DB2_819 : Bool := TRUE;   // Error messages / Signalisations de défaut
      User33_DB2_820 : Bool := TRUE;   // Error messages / Signalisations de défaut
      User33_DB2_821 : Bool := TRUE;   // Error messages / Signalisations de défaut
      User33_DB2_822 : Bool := FALSE;   // Operating messages / Signalisations d'état
      User33_DB2_823 : Bool := FALSE;   // Operating messages / Signalisations d'état
      User33_DB2_824 : Bool := FALSE;   // Operating messages / Signalisations d'état
      User33_DB2_825 : Bool := FALSE;   // Operating messages / Signalisations d'état
      User34_DB2_826 : Bool := TRUE;   // UserDataArea 34, DB2.DBB826; error messages / UserDataArea 34, DB2.DBB826 ; signalisations de défaut
      User34_DB2_827 : Bool := TRUE;   // Error messages / Signalisations de défaut
      User34_DB2_828 : Bool := TRUE;   // Error messages / Signalisations de défaut
      User34_DB2_829 : Bool := TRUE;   // Error messages / Signalisations de défaut
      User34_DB2_830 : Bool := FALSE;   // Operating messages / Signalisations d'état
      User34_DB2_831 : Bool := FALSE;   // Operating messages / Signalisations d'état
      User34_DB2_832 : Bool := FALSE;   // Operating messages / Signalisations d'état
      User34_DB2_833 : Bool := FALSE;   // Operating messages / Signalisations d'état
      User35_DB2_834 : Bool := TRUE;   // UserDataArea 35, DB2.DBB834; error messages / UserDataArea 35, DB2.DBB834 ; signalisations de défaut
      User35_DB2_835 : Bool := TRUE;   // Error messages / Signalisations de défaut
      User35_DB2_836 : Bool := TRUE;   // Error messages / Signalisations de défaut
      User35_DB2_837 : Bool := TRUE;   // Error messages / Signalisations de défaut
      User35_DB2_838 : Bool := FALSE;   // Operating messages / Signalisations d'état
      User35_DB2_839 : Bool := FALSE;   // Operating messages / Signalisations d'état
      User35_DB2_840 : Bool := FALSE;   // Operating messages / Signalisations d'état
      User35_DB2_841 : Bool := FALSE;   // Operating messages / Signalisations d'état
      User36_DB2_842 : Bool := TRUE;   // UserDataArea 36, DB2.DBB842; error messages / UserDataArea 36, DB2.DBB842 ; signalisations de défaut
      User36_DB2_843 : Bool := TRUE;   // Error messages / Signalisations de défaut
      User36_DB2_844 : Bool := TRUE;   // Error messages / Signalisations de défaut
      User36_DB2_845 : Bool := TRUE;   // Error messages / Signalisations de défaut
      User36_DB2_846 : Bool := FALSE;   // Operating messages / Signalisations d'état
      User36_DB2_847 : Bool := FALSE;   // Operating messages / Signalisations d'état
      User36_DB2_848 : Bool := FALSE;   // Operating messages / Signalisations d'état
      User36_DB2_849 : Bool := FALSE;   // Operating messages / Signalisations d'état
      User37_DB2_850 : Bool := TRUE;   // UserDataArea 37, DB2.DBB850; error messages / UserDataArea 37, DB2.DBB850 ; signalisations de défaut
      User37_DB2_851 : Bool := TRUE;   // Error messages / Signalisations de défaut
      User37_DB2_852 : Bool := TRUE;   // Error messages / Signalisations de défaut
      User37_DB2_853 : Bool := TRUE;   // Error messages / Signalisations de défaut
      User37_DB2_854 : Bool := FALSE;   // Operating messages / Signalisations d'état
      User37_DB2_855 : Bool := FALSE;   // Operating messages / Signalisations d'état
      User37_DB2_856 : Bool := FALSE;   // Operating messages / Signalisations d'état
      User37_DB2_857 : Bool := FALSE;   // Operating messages / Signalisations d'état
      User38_DB2_858 : Bool := TRUE;   // UserDataArea 38, DB2.DBB858; error messages / UserDataArea 38, DB2.DBB858 ; signalisations de défaut
      User38_DB2_859 : Bool := TRUE;   // Error messages / Signalisations de défaut
      User38_DB2_860 : Bool := TRUE;   // Error messages / Signalisations de défaut
      User38_DB2_861 : Bool := TRUE;   // Error messages / Signalisations de défaut
      User38_DB2_862 : Bool := FALSE;   // Operating messages / Signalisations d'état
      User38_DB2_863 : Bool := FALSE;   // Operating messages / Signalisations d'état
      User38_DB2_864 : Bool := FALSE;   // Operating messages / Signalisations d'état
      User38_DB2_865 : Bool := FALSE;   // Operating messages / Signalisations d'état
      User39_DB2_866 : Bool := TRUE;   // UserDataArea 39, DB2.DBB866; error messages / UserDataArea 39, DB2.DBB866 ; signalisations de défaut
      User39_DB2_867 : Bool := TRUE;   // Error messages / Signalisations de défaut
      User39_DB2_868 : Bool := TRUE;   // Error messages / Signalisations de défaut
      User39_DB2_869 : Bool := TRUE;   // Error messages / Signalisations de défaut
      User39_DB2_870 : Bool := FALSE;   // Operating messages / Signalisations d'état
      User39_DB2_871 : Bool := FALSE;   // Operating messages / Signalisations d'état
      User39_DB2_872 : Bool := FALSE;   // Operating messages / Signalisations d'état
      User39_DB2_873 : Bool := FALSE;   // Operating messages / Signalisations d'état
      User40_DB2_874 : Bool := TRUE;   // UserDataArea 40, DB2.DBB874; error messages / UserDataArea 40, DB2.DBB874 ; signalisations de défaut
      User40_DB2_875 : Bool := TRUE;   // Error messages / Signalisations de défaut
      User40_DB2_876 : Bool := TRUE;   // Error messages / Signalisations de défaut
      User40_DB2_877 : Bool := TRUE;   // Error messages / Signalisations de défaut
      User40_DB2_878 : Bool := FALSE;   // Operating messages / Signalisations d'état
      User40_DB2_879 : Bool := FALSE;   // Operating messages / Signalisations d'état
      User40_DB2_880 : Bool := FALSE;   // Operating messages / Signalisations d'état
      User40_DB2_881 : Bool := FALSE;   // Operating messages / Signalisations d'état
      User41_DB2_882 : Bool := TRUE;   // UserDataArea 41, DB2.DBB882; error messages / UserDataArea 41, DB2.DBB882 ; signalisations de défaut
      User41_DB2_883 : Bool := TRUE;   // Error messages / Signalisations de défaut
      User41_DB2_884 : Bool := TRUE;   // Error messages / Signalisations de défaut
      User41_DB2_885 : Bool := TRUE;   // Error messages / Signalisations de défaut
      User41_DB2_886 : Bool := FALSE;   // Operating messages / Signalisations d'état
      User41_DB2_887 : Bool := FALSE;   // Operating messages / Signalisations d'état
      User41_DB2_888 : Bool := FALSE;   // Operating messages / Signalisations d'état
      User41_DB2_889 : Bool := FALSE;   // Operating messages / Signalisations d'état
      User42_DB2_890 : Bool := TRUE;   // UserDataArea 42, DB2.DBB890; error messages / UserDataArea 42, DB2.DBB890 ; signalisations de défaut
      User42_DB2_891 : Bool := TRUE;   // Error messages / Signalisations de défaut
      User42_DB2_892 : Bool := TRUE;   // Error messages / Signalisations de défaut
      User42_DB2_893 : Bool := TRUE;   // Error messages / Signalisations de défaut
      User42_DB2_894 : Bool := FALSE;   // Operating messages / Signalisations d'état
      User42_DB2_895 : Bool := FALSE;   // Operating messages / Signalisations d'état
      User42_DB2_896 : Bool := FALSE;   // Operating messages / Signalisations d'état
      User42_DB2_897 : Bool := FALSE;   // Operating messages / Signalisations d'état
      User43_DB2_898 : Bool := TRUE;   // UserDataArea 43, DB2.DBB898; error messages / UserDataArea 43, DB2.DBB898 ; signalisations de défaut
      User43_DB2_899 : Bool := TRUE;   // Error messages / Signalisations de défaut
      User43_DB2_900 : Bool := TRUE;   // Error messages / Signalisations de défaut
      User43_DB2_901 : Bool := TRUE;   // Error messages / Signalisations de défaut
      User43_DB2_902 : Bool := FALSE;   // Operating messages / Signalisations d'état
      User43_DB2_903 : Bool := FALSE;   // Operating messages / Signalisations d'état
      User43_DB2_904 : Bool := FALSE;   // Operating messages / Signalisations d'état
      User43_DB2_905 : Bool := FALSE;   // Operating messages / Signalisations d'état
      User44_DB2_906 : Bool := TRUE;   // UserDataArea 44, DB2.DBB906; error messages / UserDataArea 44, DB2.DBB906 ; signalisations de défaut
      User44_DB2_907 : Bool := TRUE;   // Error messages / Signalisations de défaut
      User44_DB2_908 : Bool := TRUE;   // Error messages / Signalisations de défaut
      User44_DB2_909 : Bool := TRUE;   // Error messages / Signalisations de défaut
      User44_DB2_910 : Bool := FALSE;   // Operating messages / Signalisations d'état
      User44_DB2_911 : Bool := FALSE;   // Operating messages / Signalisations d'état
      User44_DB2_912 : Bool := FALSE;   // Operating messages / Signalisations d'état
      User44_DB2_913 : Bool := FALSE;   // Operating messages / Signalisations d'état
      User45_DB2_914 : Bool := TRUE;   // UserDataArea 45, DB2.DBB914; error messages / UserDataArea 45, DB2.DBB914 ; signalisations de défaut
      User45_DB2_915 : Bool := TRUE;   // Error messages / Signalisations de défaut
      User45_DB2_916 : Bool := TRUE;   // Error messages / Signalisations de défaut
      User45_DB2_917 : Bool := TRUE;   // Error messages / Signalisations de défaut
      User45_DB2_918 : Bool := FALSE;   // Operating messages / Signalisations d'état
      User45_DB2_919 : Bool := FALSE;   // Operating messages / Signalisations d'état
      User45_DB2_920 : Bool := FALSE;   // Operating messages / Signalisations d'état
      User45_DB2_921 : Bool := FALSE;   // Operating messages / Signalisations d'état
      User46_DB2_922 : Bool := TRUE;   // UserDataArea 46, DB2.DBB922; error messages / UserDataArea 46, DB2.DBB922 ; signalisations de défaut
      User46_DB2_923 : Bool := TRUE;   // Error messages / Signalisations de défaut
      User46_DB2_924 : Bool := TRUE;   // Error messages / Signalisations de défaut
      User46_DB2_925 : Bool := TRUE;   // Error messages / Signalisations de défaut
      User46_DB2_926 : Bool := FALSE;   // Operating messages / Signalisations d'état
      User46_DB2_927 : Bool := FALSE;   // Operating messages / Signalisations d'état
      User46_DB2_928 : Bool := FALSE;   // Operating messages / Signalisations d'état
      User46_DB2_929 : Bool := FALSE;   // Operating messages / Signalisations d'état
      User47_DB2_930 : Bool := TRUE;   // UserDataArea 47, DB2.DBB930; error messages / UserDataArea 47, DB2.DBB930 ; signalisations de défaut
      User47_DB2_931 : Bool := TRUE;   // Error messages / Signalisations de défaut
      User47_DB2_932 : Bool := TRUE;   // Error messages / Signalisations de défaut
      User47_DB2_933 : Bool := TRUE;   // Error messages / Signalisations de défaut
      User47_DB2_934 : Bool := FALSE;   // Operating messages / Signalisations d'état
      User47_DB2_935 : Bool := FALSE;   // Operating messages / Signalisations d'état
      User47_DB2_936 : Bool := FALSE;   // Operating messages / Signalisations d'état
      User47_DB2_937 : Bool := FALSE;   // Operating messages / Signalisations d'état
      User48_DB2_938 : Bool := TRUE;   // UserDataArea 48, DB2.DBB938; error messages / UserDataArea 48, DB2.DBB938 ; signalisations de défaut
      User48_DB2_939 : Bool := TRUE;   // Error messages / Signalisations de défaut
      User48_DB2_940 : Bool := TRUE;   // Error messages / Signalisations de défaut
      User48_DB2_941 : Bool := TRUE;   // Error messages / Signalisations de défaut
      User48_DB2_942 : Bool := FALSE;   // Operating messages / Signalisations d'état
      User48_DB2_943 : Bool := FALSE;   // Operating messages / Signalisations d'état
      User48_DB2_944 : Bool := FALSE;   // Operating messages / Signalisations d'état
      User48_DB2_945 : Bool := FALSE;   // Operating messages / Signalisations d'état
      User49_DB2_946 : Bool := TRUE;   // UserDataArea 49, DB2.DBB946; error messages / UserDataArea 49, DB2.DBB946 ; signalisations de défaut
      User49_DB2_947 : Bool := TRUE;   // Error messages / Signalisations de défaut
      User49_DB2_948 : Bool := TRUE;   // Error messages / Signalisations de défaut
      User49_DB2_949 : Bool := TRUE;   // Error messages / Signalisations de défaut
      User49_DB2_950 : Bool := FALSE;   // Operating messages / Signalisations d'état
      User49_DB2_951 : Bool := FALSE;   // Operating messages / Signalisations d'état
      User49_DB2_952 : Bool := FALSE;   // Operating messages / Signalisations d'état
      User49_DB2_953 : Bool := FALSE;   // Operating messages / Signalisations d'état
      User50_DB2_954 : Bool := TRUE;   // UserDataArea 50, DB2.DBB954; error messages / UserDataArea 50, DB2.DBB954 ; signalisations de défaut
      User50_DB2_955 : Bool := TRUE;   // Error messages / Signalisations de défaut
      User50_DB2_956 : Bool := TRUE;   // Error messages / Signalisations de défaut
      User50_DB2_957 : Bool := TRUE;   // Error messages / Signalisations de défaut
      User50_DB2_958 : Bool := FALSE;   // Operating messages / Signalisations d'état
      User50_DB2_959 : Bool := FALSE;   // Operating messages / Signalisations d'état
      User50_DB2_960 : Bool := FALSE;   // Operating messages / Signalisations d'état
      User50_DB2_961 : Bool := FALSE;   // Operating messages / Signalisations d'état
      User51_DB2_962 : Bool := TRUE;   // UserDataArea 51, DB2.DBB962; error messages / UserDataArea 51, DB2.DBB962 ; signalisations de défaut
      User51_DB2_963 : Bool := TRUE;   // Error messages / Signalisations de défaut
      User51_DB2_964 : Bool := TRUE;   // Error messages / Signalisations de défaut
      User51_DB2_965 : Bool := TRUE;   // Error messages / Signalisations de défaut
      User51_DB2_966 : Bool := FALSE;   // Operating messages / Signalisations d'état
      User51_DB2_967 : Bool := FALSE;   // Operating messages / Signalisations d'état
      User51_DB2_968 : Bool := FALSE;   // Operating messages / Signalisations d'état
      User51_DB2_969 : Bool := FALSE;   // Operating messages / Signalisations d'état
      User52_DB2_970 : Bool := TRUE;   // UserDataArea 52, DB2.DBB970; error messages / UserDataArea 52, DB2.DBB970 ; signalisations de défaut
      User52_DB2_971 : Bool := TRUE;   // Error messages / Signalisations de défaut
      User52_DB2_972 : Bool := TRUE;   // Error messages / Signalisations de défaut
      User52_DB2_973 : Bool := TRUE;   // Error messages / Signalisations de défaut
      User52_DB2_974 : Bool := FALSE;   // Operating messages / Signalisations d'état
      User52_DB2_975 : Bool := FALSE;   // Operating messages / Signalisations d'état
      User52_DB2_976 : Bool := FALSE;   // Operating messages / Signalisations d'état
      User52_DB2_977 : Bool := FALSE;   // Operating messages / Signalisations d'état
      User53_DB2_978 : Bool := TRUE;   // UserDataArea 53, DB2.DBB978; error messages / UserDataArea 53, DB2.DBB978 ; signalisations de défaut
      User53_DB2_979 : Bool := TRUE;   // Error messages / Signalisations de défaut
      User53_DB2_980 : Bool := TRUE;   // Error messages / Signalisations de défaut
      User53_DB2_981 : Bool := TRUE;   // Error messages / Signalisations de défaut
      User53_DB2_982 : Bool := FALSE;   // Operating messages / Signalisations d'état
      User53_DB2_983 : Bool := FALSE;   // Operating messages / Signalisations d'état
      User53_DB2_984 : Bool := FALSE;   // Operating messages / Signalisations d'état
      User53_DB2_985 : Bool := FALSE;   // Operating messages / Signalisations d'état
      User54_DB2_986 : Bool := TRUE;   // UserDataArea 54, DB2.DBB986; error messages / UserDataArea 54, DB2.DBB986 ; signalisations de défaut
      User54_DB2_987 : Bool := TRUE;   // Error messages / Signalisations de défaut
      User54_DB2_988 : Bool := TRUE;   // Error messages / Signalisations de défaut
      User54_DB2_989 : Bool := TRUE;   // Error messages / Signalisations de défaut
      User54_DB2_990 : Bool := FALSE;   // Operating messages / Signalisations d'état
      User54_DB2_991 : Bool := FALSE;   // Operating messages / Signalisations d'état
      User54_DB2_992 : Bool := FALSE;   // Operating messages / Signalisations d'état
      User54_DB2_993 : Bool := FALSE;   // Operating messages / Signalisations d'état
      User55_DB2_994 : Bool := TRUE;   // UserDataArea 55, DB2.DBB994; error messages / UserDataArea 55, DB2.DBB994 ; signalisations de défaut
      User55_DB2_995 : Bool := TRUE;   // Error messages / Signalisations de défaut
      User55_DB2_996 : Bool := TRUE;   // Error messages / Signalisations de défaut
      User55_DB2_997 : Bool := TRUE;   // Error messages / Signalisations de défaut
      User55_DB2_998 : Bool := FALSE;   // Operating messages / Signalisations d'état
      User55_DB2_999 : Bool := FALSE;   // Operating messages / Signalisations d'état
      User55_DB2_1000 : Bool := FALSE;   // Operating messages / Signalisations d'état
      User55_DB2_1001 : Bool := FALSE;   // Operating messages / Signalisations d'état
      User56_DB2_1002 : Bool := TRUE;   // UserDataArea 56, DB2.DBB1002; error messages / UserDataArea 56, DB2.DBB1002 ; signalisations de défaut
      User56_DB2_1003 : Bool := TRUE;   // Error messages / Signalisations de défaut
      User56_DB2_1004 : Bool := TRUE;   // Error messages / Signalisations de défaut
      User56_DB2_1005 : Bool := TRUE;   // Error messages / Signalisations de défaut
      User56_DB2_1006 : Bool := FALSE;   // Operating messages / Signalisations d'état
      User56_DB2_1007 : Bool := FALSE;   // Operating messages / Signalisations d'état
      User56_DB2_1008 : Bool := FALSE;   // Operating messages / Signalisations d'état
      User56_DB2_1009 : Bool := FALSE;   // Operating messages / Signalisations d'état
      User57_DB2_1010 : Bool := TRUE;   // UserDataArea 57, DB2.DBB1010; error messages / UserDataArea 57, DB2.DBB1010 ; signalisations de défaut
      User57_DB2_1011 : Bool := TRUE;   // Error messages / Signalisations de défaut
      User57_DB2_1012 : Bool := TRUE;   // Error messages / Signalisations de défaut
      User57_DB2_1013 : Bool := TRUE;   // Error messages / Signalisations de défaut
      User57_DB2_1014 : Bool := FALSE;   // Operating messages / Signalisations d'état
      User57_DB2_1015 : Bool := FALSE;   // Operating messages / Signalisations d'état
      User57_DB2_1016 : Bool := FALSE;   // Operating messages / Signalisations d'état
      User57_DB2_1017 : Bool := FALSE;   // Operating messages / Signalisations d'état
      User58_DB2_1018 : Bool := TRUE;   // UserDataArea 58, DB2.DBB1018; error messages / UserDataArea 58, DB2.DBB1018 ; signalisations de défaut
      User58_DB2_1019 : Bool := TRUE;   // Error messages / Signalisations de défaut
      User58_DB2_1020 : Bool := TRUE;   // Error messages / Signalisations de défaut
      User58_DB2_1021 : Bool := TRUE;   // Error messages / Signalisations de défaut
      User58_DB2_1022 : Bool := FALSE;   // Operating messages / Signalisations d'état
      User58_DB2_1023 : Bool := FALSE;   // Operating messages / Signalisations d'état
      User58_DB2_1024 : Bool := FALSE;   // Operating messages / Signalisations d'état
      User58_DB2_1025 : Bool := FALSE;   // Operating messages / Signalisations d'état
      User59_DB2_1026 : Bool := TRUE;   // UserDataArea 59, DB2.DBB1026; error messages / UserDataArea 59, DB2.DBB1026 ; signalisations de défaut
      User59_DB2_1027 : Bool := TRUE;   // Error messages / Signalisations de défaut
      User59_DB2_1028 : Bool := TRUE;   // Error messages / Signalisations de défaut
      User59_DB2_1029 : Bool := TRUE;   // Error messages / Signalisations de défaut
      User59_DB2_1030 : Bool := FALSE;   // Operating messages / Signalisations d'état
      User59_DB2_1031 : Bool := FALSE;   // Operating messages / Signalisations d'état
      User59_DB2_1032 : Bool := FALSE;   // Operating messages / Signalisations d'état
      User59_DB2_1033 : Bool := FALSE;   // Operating messages / Signalisations d'état
      User60_DB2_1034 : Bool := TRUE;   // UserDataArea 60, DB2.DBB1034; error messages / UserDataArea 60, DB2.DBB1034 ; signalisations de défaut
      User60_DB2_1035 : Bool := TRUE;   // Error messages / Signalisations de défaut
      User60_DB2_1036 : Bool := TRUE;   // Error messages / Signalisations de défaut
      User60_DB2_1037 : Bool := TRUE;   // Error messages / Signalisations de défaut
      User60_DB2_1038 : Bool := FALSE;   // Operating messages / Signalisations d'état
      User60_DB2_1039 : Bool := FALSE;   // Operating messages / Signalisations d'état
      User60_DB2_1040 : Bool := FALSE;   // Operating messages / Signalisations d'état
      User60_DB2_1041 : Bool := FALSE;   // Operating messages / Signalisations d'état
      User61_DB2_1042 : Bool := TRUE;   // UserDataArea 61, DB2.DBB1042; error messages / UserDataArea 61, DB2.DBB1042 ; signalisations de défaut
      User61_DB2_1043 : Bool := TRUE;   // Error messages / Signalisations de défaut
      User61_DB2_1044 : Bool := TRUE;   // Error messages / Signalisations de défaut
      User61_DB2_1045 : Bool := TRUE;   // Error messages / Signalisations de défaut
      User61_DB2_1046 : Bool := FALSE;   // Operating messages / Signalisations d'état
      User61_DB2_1047 : Bool := FALSE;   // Operating messages / Signalisations d'état
      User61_DB2_1048 : Bool := FALSE;   // Operating messages / Signalisations d'état
      User61_DB2_1049 : Bool := FALSE;   // Operating messages / Signalisations d'état
      User62_DB2_1050 : Bool := TRUE;   // UserDataArea 62, DB2.DBB1050; error messages / UserDataArea 62, DB2.DBB1050 ; signalisations de défaut
      User62_DB2_1051 : Bool := TRUE;   // Error messages / Signalisations de défaut
      User62_DB2_1052 : Bool := TRUE;   // Error messages / Signalisations de défaut
      User62_DB2_1053 : Bool := TRUE;   // Error messages / Signalisations de défaut
      User62_DB2_1054 : Bool := FALSE;   // Operating messages / Signalisations d'état
      User62_DB2_1055 : Bool := FALSE;   // Operating messages / Signalisations d'état
      User62_DB2_1056 : Bool := FALSE;   // Operating messages / Signalisations d'état
      User62_DB2_1057 : Bool := FALSE;   // Operating messages / Signalisations d'état
      User63_DB2_1058 : Bool := TRUE;   // UserDataArea 63, DB2.DBB1058; error messages / UserDataArea 63, DB2.DBB1058 ; signalisations de défaut
      User63_DB2_1059 : Bool := TRUE;   // Error messages / Signalisations de défaut
      User63_DB2_1060 : Bool := TRUE;   // Error messages / Signalisations de défaut
      User63_DB2_1061 : Bool := TRUE;   // Error messages / Signalisations de défaut
      User63_DB2_1062 : Bool := FALSE;   // Operating messages / Signalisations d'état
      User63_DB2_1063 : Bool := FALSE;   // Operating messages / Signalisations d'état
      User63_DB2_1064 : Bool := FALSE;   // Operating messages / Signalisations d'état
      User63_DB2_1065 : Bool := FALSE;   // Operating messages / Signalisations d'état
   END_VAR
BEGIN
END_DATA_BLOCK
